(* IEC 61131-3 sources: Roaster_s7-200/I2C_test/build, 2 files *)

(* ---- plc.st ---- *)
TYPE
  LOGLEVEL : (CRITICAL, WARNING, INFO, DEBUG) := INFO;
END_TYPE

FUNCTION_BLOCK LOGGER
  VAR_INPUT
    TRIG : BOOL;
    MSG : STRING;
    LEVEL : LOGLEVEL := INFO;
  END_VAR
  VAR
    TRIG0 : BOOL;
  END_VAR

  IF TRIG AND NOT TRIG0 THEN
  {{
   LogMessage(GetFbVar(LEVEL),(char*)GetFbVar(MSG, .body),GetFbVar(MSG, .len));
  }}
  END_IF;
  TRIG0:=TRIG;
END_FUNCTION_BLOCK

FUNCTION_BLOCK python_eval
  VAR_INPUT
    TRIG : BOOL;
    CODE : STRING;
  END_VAR
  VAR_OUTPUT
    ACK : BOOL;
    RESULT : STRING;
  END_VAR
  VAR
    STATE : DWORD;
    BUFFER : STRING;
    PREBUFFER : STRING;
    TRIGM1 : BOOL;
    TRIGGED : BOOL;
  END_VAR

  {extern void __PythonEvalFB(int, PYTHON_EVAL*);__PythonEvalFB(0, data__);}
END_FUNCTION_BLOCK

FUNCTION_BLOCK python_poll
  VAR_INPUT
    TRIG : BOOL;
    CODE : STRING;
  END_VAR
  VAR_OUTPUT
    ACK : BOOL;
    RESULT : STRING;
  END_VAR
  VAR
    STATE : DWORD;
    BUFFER : STRING;
    PREBUFFER : STRING;
    TRIGM1 : BOOL;
    TRIGGED : BOOL;
  END_VAR

  {extern void __PythonEvalFB(int, PYTHON_EVAL*);__PythonEvalFB(1,(PYTHON_EVAL*)(void*)data__);}
END_FUNCTION_BLOCK

FUNCTION_BLOCK python_gear
  VAR_INPUT
    N : UINT;
    TRIG : BOOL;
    CODE : STRING;
  END_VAR
  VAR_OUTPUT
    ACK : BOOL;
    RESULT : STRING;
  END_VAR
  VAR
    py_eval : python_eval;
    COUNTER : UINT;
    _TMP_ADD10_OUT : UINT;
    _TMP_EQ13_OUT : BOOL;
    _TMP_SEL15_OUT : UINT;
    _TMP_AND7_OUT : BOOL;
  END_VAR

  _TMP_ADD10_OUT := ADD(COUNTER, 1);
  _TMP_EQ13_OUT := EQ(N, _TMP_ADD10_OUT);
  _TMP_SEL15_OUT := SEL(_TMP_EQ13_OUT, _TMP_ADD10_OUT, 0);
  COUNTER := _TMP_SEL15_OUT;
  _TMP_AND7_OUT := AND(_TMP_EQ13_OUT, TRIG);
  py_eval(TRIG := _TMP_AND7_OUT, CODE := CODE);
  ACK := py_eval.ACK;
  RESULT := py_eval.RESULT;
END_FUNCTION_BLOCK

PROGRAM get_temp
  VAR
    I2C_AHT200 : I2C_AHT20;
    sck : INT := 5;
    sda : INT := 4;
    temp : REAL;
    RH0 : REAL;
  END_VAR

  I2C_AHT200(EN := TRUE, SCK_PIN := sck, SDA_PIN := sda);
  IF I2C_AHT200.ENO THEN
      temp := I2C_AHT200.TEMP;
  END_IF;
  IF I2C_AHT200.ENO THEN
      RH0 := I2C_AHT200.RH;
  END_IF;
END_PROGRAM

PROGRAM main
  VAR
    in : BOOL;
    out : BOOL;
  END_VAR

  out := in;
END_PROGRAM

CONFIGURATION Config0

  RESOURCE Res0 ON PLC
    TASK task0(INTERVAL := T#20ms,PRIORITY := 0);
    TASK task1(INTERVAL := T#1000ms,PRIORITY := 1);
    PROGRAM instance0 WITH task0 : main;
    PROGRAM instance1 WITH task1 : get_temp;
  END_RESOURCE
END_CONFIGURATION

(* ---- generated_plc.st ---- *)
PROGRAM get_temp
  VAR
    I2C_AHT200 : I2C_AHT20;
    sck : INT := 5;
    sda : INT := 4;
    temp : REAL;
    RH0 : REAL;
  END_VAR

  I2C_AHT200(EN := TRUE, SCK_PIN := sck, SDA_PIN := sda);
  IF I2C_AHT200.ENO THEN
      temp := I2C_AHT200.TEMP;
  END_IF;
  IF I2C_AHT200.ENO THEN
      RH0 := I2C_AHT200.RH;
  END_IF;
END_PROGRAM

PROGRAM main
  VAR
    in AT %IX0.2 : BOOL;
    out AT %QX0.2 : BOOL;
  END_VAR

  out := in;
END_PROGRAM

CONFIGURATION Config0

  RESOURCE Res0 ON PLC
    TASK task0(INTERVAL := T#20ms,PRIORITY := 0);
    TASK task1(INTERVAL := T#1000ms,PRIORITY := 1);
    PROGRAM instance0 WITH task0 : main;
    PROGRAM instance1 WITH task1 : get_temp;
  END_RESOURCE
END_CONFIGURATION
